{attribute 'linkalways'} 
{attribute 'no_explicit_call' := 'This FB is a CLASS and must be accessed using methods or properties'}
{attribute 'enable_dynamic_creation'}
FUNCTION_BLOCK Node_F_VN_GetAt_INT EXTENDS VisionNode
VAR
    ipContainer : _ITcVnContainer;
    nElement : _INT(0);
    nIndex : _ULINT(0);
    hrPrev : _HRESULT(S_OK);
    hresult : _HRESULT(S_OK);
END_VAR

METHOD PUBLIC  Clone : I_Node
VAR
	pNode : POINTER TO Node_F_VN_GetAt_INT;
END_VAR
pNode := __NEW(Node_F_VN_GetAt_INT);
Clone := pNode^;
END_METHOD

METHOD FB_init : BOOL
VAR_INPUT
	bInitRetains : BOOL; // if TRUE, the retain variables are initialized (warm start / cold start)
	bInCopyCode : BOOL;  // if TRUE, the instance afterwards gets moved into the copy code (online change)
END_VAR
AddInput('ipContainer', ipContainer);
AddParameter('nIndex', nIndex);
AddInput('hrPrev', hrPrev);
AddOutput('nElement', nElement);
AddOutput('hresult',hresult);
END_METHOD

METHOD PROTECTED OnExecute
hresult.Value := F_VN_GetAt_INT(
    ipContainer := ipContainer.Value,
    nElement := nElement.Value,
    nIndex := nIndex.Value,
    hrPrev:= hrPrev.Value);
END_METHOD

METHOD PUBLIC PreExecutionCheck
VAR_INPUT
	Check : I_PreExecutionChecks;
END_VAR
Check.IsTrue(ipContainer.IsValid, 'ipContainer must be a valid container');
Check.IsTrue(ipContainer.IsType(TC_GLOBAL_CONST_LIST.ContainerType_Vector_INT), 'ipContainer contains incorrect type');
END_METHOD

END_FUNCTION_BLOCK

(* stored: Version 1.1.0.1, ProductVersion 3.1.4026.13
   POU Node_F_VN_GetAt_INT: Id {0ce6958f-f8a7-43e8-80b0-9b01f90277a9}, SpecialFunc None
   Folder Constructor: Id {6027bc70-3675-4036-b501-132e06b87159}
   Method Clone: Id {2e1b0f75-9196-40cf-9524-a52eac4c71b7}
   Method FB_init: Id {cc5da3be-615c-4455-b6d4-e8c7361b67a2}
   Method OnExecute: Id {1bb48613-2ae1-4e36-a46e-a85a66b821cd}
   Method PreExecutionCheck: Id {9d407a86-40c8-45e6-84a7-3f2efa23c31d} *)
